KUKA KRL program: D15_main.src, D15_main.dat

--- D15_main.src ---
&ACCESS RVP1
&REL 7
&COMMENT SbtComm001 Main
&PARAM EDITMASK = *
&PARAM DISKPATH = KRC:\R1\Program\SbtComm001Main\D
DEF D15_main( )
;***********************************************************
;
; Copyright 2018 - 2025 speedbot All Rights reserved.
;
; File Name: mixsort_main.DAT
;
; Description:
;   Language             ==   Krl for KUKA ROBOT
;   Date                 ==   2022 - 06 - 27
;   Modification Data    ==   2025 - 02 - 10
;
; Author: speedbot
;
; Version: 1.1
;***********************************************************
;FOLD INI;%{PE}
    ;FOLD BASISTECH INI
        GLOBAL INTERRUPT DECL 3 WHEN $STOPMESS==TRUE DO IR_STOPM ( )
        INTERRUPT ON 3
        BAS (#INITMOV,0 )
    ;ENDFOLD (BASISTECH INI)
    ;FOLD USER INI
        ;Make your modifications here

    ;ENDFOLD (USER INI)
;ENDFOLD (INI)
;FOLD Basic.Override IN Override: 30  ;%{PE}
override_(30)
;ENDFOLD
;FOLD PLC.Pounce ;%{PE}
pounce_()
;ENDFOLD
D15_DCD_PICK()
D15_DCD_DROP()
;FOLD PLC.MoveToHome ;%{PE}
move_to_home_()
;ENDFOLD
END

--- D15_main.dat ---
&ACCESS RVP1
&REL 7
&COMMENT SbtComm001 Main
&PARAM EDITMASK = *
&PARAM DISKPATH = KRC:\R1\Program\SbtComm001Main\D
DEFDAT  D15_MAIN
;***********************************************************
;
; Copyright 2018 - 2025 speedbot All Rights reserved.
;
; File Name: mixsort_main.DAT
;
; Description:
;   Language             ==   Krl for KUKA ROBOT
;   Date                 ==   2022 - 06 - 27
;   Modification Data    ==   2025 - 02 - 10
;
; Author: speedbot
;
; Version: 1.1
;***********************************************************
;FOLD EXTERNAL DECLARATIONS;%{PE}%MKUKATPBASIS,%CEXT,%VCOMMON,%P
;FOLD BASISTECH EXT;%{PE}%MKUKATPBASIS,%CEXT,%VEXT,%P
EXT  BAS (BAS_COMMAND  :IN,REAL  :IN )

DECL INT SUCCESS
;ENDFOLD (BASISTECH EXT)
;FOLD USER EXT;%{E}%MKUKATPUSER,%CEXT,%VEXT,%P
;Make your modifications here

;ENDFOLD (USER EXT)
;ENDFOLD (EXTERNAL DECLARATIONS)

DECL MODULEPARAM_T LAST_TP_PARAMS={PARAMS[] "BASIC.OVERRIDESPEED=30          "}
ENDDAT
